TYPE Mat5d : ARRAY[1..5, 1..5] OF LREAL; END_TYPE

(* stored: Version 1.1.0.1, ProductVersion 3.1.4024.12
   DUT Mat5d: Id {e4d97ec9-57d0-4d03-a160-cd23c2d3a041} *)
